PROGRAM Modbus_ReadInputs
VAR
	bReadInputs : 	BOOL;
	tReadInputs	: 	TON;
	ReadInputs	: FB_MBReadInputs;

END_VAR

//Modbus read inputs function.
tReadInputs(IN:= NOT ReadInputs.bBusy, PT:= T#10MS , Q=> bReadInputs, ET=> );

ReadInputs(
	sIPAddr:= '127.0.0.1', 
	nTCPPort:= 505, 
	nUnitID:= 255, 
	nQuantity:= 14, 
	nMBAddr:= 0, 
	cbLength:= SIZEOF(InputArea), 
	pDestAddr:= ADR(InputArea), 
	bExecute:= bReadInputs, 
	tTimeout:= T#1S, 
	bBusy=> , 
	bError=> , 
	nErrId=> , 
	cbRead=> );

END_PROGRAM

(* stored: Version 1.1.0.1, ProductVersion 3.1.4024.6
   POU Modbus_ReadInputs: Id {afbc1203-c214-431a-8ef8-de537497029b}, SpecialFunc None *)
